PROGRAM PRG_TEST_ThreeDOF_robot
VAR
	fb_RC_Servo_Test : FB_RC_Servo_Test;
	fb_Sequence_Recorder : FB_Sequence_Recorder_Test;
	fb_Clamp_INT_Test : FB_Clamp_INT_Test;
END_VAR

TcUnit.RUN();

END_PROGRAM

(* stored: Version 1.1.0.1, ProductVersion 3.1.4024.13
   POU PRG_TEST_ThreeDOF_robot: Id {e4d7c900-4ddd-4d6a-8b55-ef2e1fbec25d}, SpecialFunc None *)
